
// ===== library: MasterCopy "Copy of Program blocks in gw_user_management" =====

// folder: gw_user_management

DATA_BLOCK "db_gw_user_logon"   // DB900
{ S7_Optimized_Access := 'TRUE' }
VERSION : 0.1
   VAR
      system : "udt_gw_user_management";
   END_VAR
BEGIN
   system.local_user_name := 'user';
   system.local_user_pwd := '1111';
   system.local_user_access_level := 400;
   system.local_technician_name := 'service';
   system.local_technician_pwd := '2222';
   system.local_technician_access_level := 600;
   system.local_admin_name := 'admin';
   system.local_admin_pwd := '43194';
   system.local_admin_access_level := 1024;
   system.logout_time := 600;
END_DATA_BLOCK

DATA_BLOCK "db_gw_faults"   // DB901
{ S7_Optimized_Access := 'TRUE' }
VERSION : 0.1
   VAR
      quitt_faults : Bool;
      fault_active : Bool;
      faults_user : "udt_gw_faults_user_management";
      quitt_faults_user : "udt_gw_faults_user_management";
   END_VAR
BEGIN
END_DATA_BLOCK

FUNCTION_BLOCK "fb_gw_user_logon"   // FB900, FBD
{ S7_Optimized_Access := 'TRUE' }
VERSION : 0.1
   VAR
      max_time_login : TON_TIME;
      logout_max_time : TON_TIME;
      timer_recovery : "udt_gw_alive_timer";
      fpos_access_level : R_TRIG;
      level_act : Bool;
   END_VAR
   VAR_TEMP
      tempLen : Int;
      i : Int;
      tempByte : Byte;
   END_VAR
BEGIN

REGION Network 1 (SCL): user name input always lower case
   IF "db_gw_user_logon".system.check_user_send OR "db_gw_user_logon".system.check_local_input_trigger THEN
       #tempLen := LEN("db_gw_user_logon".system.user_name_input);
       FOR #i := 1 TO #tempLen DO
           #tempByte := CHAR_TO_BYTE("db_gw_user_logon".system.user_name_input[#i]);
           IF #tempByte >= 65 AND #tempByte <= 90 THEN
               "db_gw_user_logon".system.user_name_input[#i] := BYTE_TO_CHAR(#tempByte + 32);
           END_IF;
       END_FOR;
   END_IF;
END_REGION

REGION Network 2 (SCL): User Verwaltung lokal / user managment local
   IF "db_gw_user_logon".system.check_local_input_trigger THEN


       IF "db_gw_user_logon".system.user_name_input = "db_gw_user_logon".system.local_user_name AND
           "db_gw_user_logon".system.password_input = "db_gw_user_logon".system.local_user_pwd THEN

           "db_gw_user_logon".system.active_user := "db_gw_user_logon".system.user_name_input;
           "db_gw_user_logon".system.access_level := "db_gw_user_logon".system.local_user_access_level;
       ELSIF
           "db_gw_user_logon".system.user_name_input = "db_gw_user_logon".system.local_technician_name AND
           "db_gw_user_logon".system.password_input = "db_gw_user_logon".system.local_technician_pwd THEN

           "db_gw_user_logon".system.active_user := "db_gw_user_logon".system.user_name_input;
           "db_gw_user_logon".system.access_level := "db_gw_user_logon".system.local_technician_access_level;
       ELSIF
           "db_gw_user_logon".system.user_name_input = "db_gw_user_logon".system.local_admin_name AND
           "db_gw_user_logon".system.password_input = "db_gw_user_logon".system.local_admin_pwd THEN

           "db_gw_user_logon".system.active_user := "db_gw_user_logon".system.user_name_input;
           "db_gw_user_logon".system.access_level := "db_gw_user_logon".system.local_admin_access_level;
       ELSE
           "db_gw_user_logon".system.active_user := '';
           "db_gw_user_logon".system.access_level := -1;
       END_IF;

       "db_gw_user_logon".system.check_local_input_trigger := FALSE;
       "db_gw_user_logon".system.user_name_input := '';
       "db_gw_user_logon".system.password_input := '';

   END_IF;
END_REGION

REGION Network 3 (SCL): user from gw-system / user managment system
   //max. time for login
   #max_time_login(IN := "db_gw_user_logon".system.check_user_send,
                   PT := T#10s);

   IF #max_time_login.Q THEN
       "db_gw_user_logon".system.chip_id_input := '';
       "db_gw_user_logon".system.check_user_send := FALSE;
       "db_gw_user_logon".system.check_user_ok := FALSE;
       "db_gw_user_logon".system.user_name_input := '';
       "db_gw_user_logon".system.password_input := '';
       "db_gw_user_logon".system.access_level := 0;
       "db_gw_faults".faults_user.fault_login_timeout := 1;
   END_IF;
END_REGION

REGION Network 4 (SCL): Abmeldezeit / logout time
   IF "db_gw_user_logon".system.access_level > 1 THEN
       #logout_max_time.PT := ("db_gw_user_logon".system.logout_time * 1000);
       IF "db_gw_user_logon".system.logout_time < 60 THEN
           "db_gw_user_logon".system.logout_time := 600;
       END_IF;
   ELSE
       "db_gw_user_logon".system.logout_time := 600;
   END_IF;

   #logout_max_time(IN := "db_gw_user_logon".system.access_level > 1,
                PT := ("db_gw_user_logon".system.logout_time * 1000));

   IF (#logout_max_time.Q OR "db_gw_user_logon".system.logout) THEN
       "db_gw_user_logon".system.active_user := '';
       "db_gw_user_logon".system.user_name_input := '';
       "db_gw_user_logon".system.password_input := '';
       "db_gw_user_logon".system.chip_id_input := '';
       "db_gw_user_logon".system.access_level := 0;
       "db_gw_user_logon".system.logout := FALSE;
   END_IF;
END_REGION

REGION Network 5 (SCL): set user access faults
   IF "db_gw_user_logon".system.check_user_ok AND "db_gw_user_logon".system.access_level < 1 THEN
       "db_gw_faults".faults_user.fault_user_access := 1;
       "db_gw_user_logon".system.check_user_ok := 0;
       "db_gw_user_logon".system.check_user_send := 0;
       "db_gw_user_logon".system.access_level := 0;
       "db_gw_user_logon".system.chip_id_input := '';
       "db_gw_user_logon".system.user_name_input := '';
       "db_gw_user_logon".system.password_input := '';
   END_IF;

   IF ("db_gw_user_logon".system.access_level < 1) AND
       "db_gw_user_logon".system.chip_id_input = '' AND
       NOT "db_gw_user_logon".system.check_local_input_trigger AND
       NOT "db_gw_user_logon".system.check_user_send THEN
       "db_gw_user_logon".system.active_user := '';
   END_IF;
END_REGION

REGION Network 6 (SCL)
   IF "db_gw_user_logon".system.check_user_send AND "db_gw_user_logon".system.check_user_ok THEN
       "db_gw_user_logon".system.chip_id_input := '';
       "db_gw_user_logon".system.check_user_send := FALSE;
       "db_gw_user_logon".system.check_user_ok := FALSE;
       "db_gw_user_logon".system.user_name_input := '';
       "db_gw_user_logon".system.password_input := '';
   END_IF;
END_REGION

REGION Network 7 (SCL): faults
   //quitt
   #level_act := "db_gw_user_logon".system.access_level > 0;
   #fpos_access_level(CLK := #level_act);

   IF "db_gw_faults".quitt_faults OR #fpos_access_level.Q THEN
       "db_gw_faults".faults_user := "db_gw_faults".quitt_faults_user;
       "db_gw_faults".quitt_faults := 0;
   END_IF;

   //faults active?
   "db_gw_faults".fault_active:="db_gw_faults".faults_user <> "db_gw_faults".quitt_faults_user;
END_REGION
END_FUNCTION_BLOCK

// ===== library: MasterCopy "udt_gw_faults_user_management" =====

TYPE "udt_gw_faults_user_management"
   STRUCT
      fault_user_access : Bool;   // fault_user_access
      fault_login_timeout : Bool;   // fault_login_timeout
   END_STRUCT;
END_TYPE

// ===== library: MasterCopy "udt_gw_user_management" =====

TYPE "udt_gw_user_management"
   STRUCT
      user_name_input : String;
      password_input : String;
      chip_id_input : String;
      access_level : Int;
      active_user : String;
      check_user_send : Bool;
      check_user_ok : Bool;
      logout : Bool;
      logout_time : DInt := 600;
      check_local_input_trigger : Bool;
      local_user_name : String := 'user';
      local_user_pwd : String := '1111';
      local_user_access_level : Int := 400;
      local_technician_name : String := 'service';
      local_technician_pwd : String := '2222';
      local_technician_access_level : Int := 600;
      local_admin_name : String := 'admin';
      local_admin_pwd : String := '43194';
      local_admin_access_level : Int := 1024;
   END_STRUCT;
END_TYPE

(* ===== HMI "HMI_RT_1" =====
connection "HMI_Verbindung_1": 

HMI tags "gw_user_management"
   "db_gw_user_logon_system" : udt_gw_user_management = PLC db_gw_user_logon.system, T500ms
   "db_gw_alive_system_alive_fault" : Bool = PLC db_gw_alive_system.alive_fault, T500ms
   "db_gw_faults_user_logon_faults_user_fault_user_access" : Bool = PLC db_gw_faults.faults_user.fault_user_access, T500ms
   "db_gw_faults_user_logon_faults_user_fault_login_timeout" : Bool = PLC db_gw_faults.faults_user.fault_login_timeout, T500ms
   "db_gw_faults_user_logon_fault_active" : Bool = PLC db_gw_faults.fault_active AT %DB1.DBX0.0, T500ms
   "db_gw_faults_user_logon_quitt_faults" : Bool = PLC db_gw_faults.quitt_faults, T500ms

discrete alarms
   2: 'User verweigert / User denied', class Alarm, trigger "db_gw_faults_user_logon_faults_user_fault_user_access" bit 0
   3: 'Timeout Login', class Alarm, trigger "db_gw_faults_user_logon_faults_user_fault_login_timeout" bit 0
   1: 'keine Verbindung zu Getzner System, nur lokale Anmeldung möglich / Getzner system unreachable - local authentication only', class Alarm, trigger "db_gw_alive_system_alive_fault" bit 0
*)

(* ===== HMI "HMI_RT_1" =====

discrete alarms
   1: 'keine Verbindung zu Getzner System, nur lokale Anmeldung möglich / Getzner system unreachable - local authentication only', class Alarm bit 0
*)

(* ===== HMI "HMI_RT_1" =====

discrete alarms
   2: 'User verweigert / User denied', class Alarm bit 0
*)

(* ===== HMI "HMI_RT_1" =====

discrete alarms
   3: 'Timeout Login', class Alarm bit 0
*)